// TIA Portal project "VISU_Registerlager_Template" (V14)

(* hardware
DEVICE "S7300/ET200M-Station_1"  S7-300 station
   slot 0: "Profilschiene_0"  Rail  6ES7 390-1***0-0AA0
   slot 2: "PLC_1"  CPU 315-2 PN/DP  6ES7 315-2EH13-0AB0  V2.6
      slot 1: "MPI/DP-Schnittstelle_1"  X1
      slot 2: "PROFINET-Schnittstelle_1"  PN-IO
         slot 1: "Port_1"  Port
*)

// ===== PLC "PLC_1"  CPU 315-2 PN/DP =====

VAR_GLOBAL   // PLC tag table "Standard-Variablentabelle"
   "CHAIN_REGISTER" AT %I10.0 : Bool;   // Förderkette Registerlager
   "REGISTER_ENGAGED" AT %I10.1 : Bool;   // Registerlager belegt
   "BELT_ENGAGED" AT %I10.2 : Bool;   // Förderband belegt
   "READ_SENSOR1" AT %I10.3 : Bool;   // Lesestation Sensor 1
   "READ_SENSOR2" AT %I10.4 : Bool;   // Lesestation Sensor 2
   "CONTROL_KEY" AT %I10.5 : Bool;   // Bedientaster
   "CHAIN_ON" AT %Q4.0 : Bool;   // Förderkette Regtisterlager an
   "LED_ON" AT %Q4.2 : Bool;   // LED an
   "BOX_NO" AT %MD1000 : DInt;   // Box-Nummer
   "BELT_ON" AT %Q4.1 : Bool;   // Förderband an
   "CON_KEY_TRIG" AT %M0.0 : Bool;   // 1 wenn Bedientaster gedrückt ist
   "CHAIN_REG_TRIG" AT %M0.1 : Bool;   // 1 wenn Sensor 3S1 aktiv wird
   "Counter_1" AT %MW1 : Int;   // Zähler für S1
   "Counter_2" AT %MW2 : Int;   // Zähler für S2
   "BELT_ENGAGED_TRIG" AT %M0.2 : Bool;   // 1 wenn der Nährungssensor aktiv ist
   "TIMER_FIN" AT %M0.3 : Bool;   // 1 wenn 15s Timer auslöst
END_VAR

ORGANIZATION_BLOCK "Main"   // OB1, FBD
TITLE = "Main Program Sweep (Cycle)"
{ S7_Optimized_Access := 'FALSE' }
VERSION : 0.1
   VAR_TEMP
      OB1_EV_CLASS : Byte;   // Bits 0-3 = 1 (Coming event), Bits 4-7 = 1 (Event class 1)
      OB1_SCAN_1 : Byte;   // 1 (Cold restart scan 1 of OB 1), 3 (Scan 2-n of OB 1)
      OB1_PRIORITY : Byte;   // Priority of OB Execution
      OB1_OB_NUMBR : Byte;   // 1 (Organization block 1, OB1)
      OB1_RESERVED_1 : Byte;   // Reserved for system
      OB1_RESERVED_2 : Byte;   // Reserved for system
      OB1_PREV_CYCLE : Int;   // Cycle time of previous OB1 scan (milliseconds)
      OB1_MIN_CYCLE : Int;   // Minimum cycle time of OB1 (milliseconds)
      OB1_MAX_CYCLE : Int;   // Maximum cycle time of OB1 (milliseconds)
      OB1_DATE_TIME : Date_And_Time;   // Date and time OB1 started
   END_VAR
   VAR_TEMP   // added for the SCL form of the ladder/FBD networks
      _w1 : Bool;
      _w2 : Bool;
   END_VAR
BEGIN

REGION Network 1: Förderkette und Förderband an
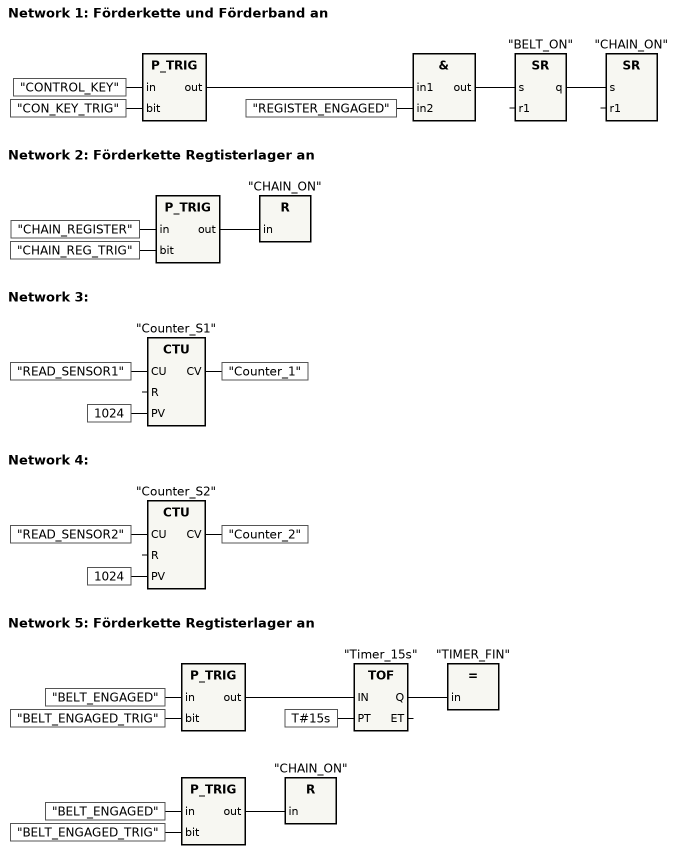
   #_w1 := "CONTROL_KEY" AND NOT "CON_KEY_TRIG";   // rising edge
   "CON_KEY_TRIG" := "CONTROL_KEY";
   IF #_w1 AND "REGISTER_ENGAGED" THEN
       "BELT_ON" := TRUE;   // SR flip-flop
   END_IF;
   IF "BELT_ON" THEN
       "CHAIN_ON" := TRUE;   // SR flip-flop
   END_IF;
END_REGION

REGION Network 2: Förderkette Regtisterlager an
   #_w1 := "CHAIN_REGISTER" AND NOT "CHAIN_REG_TRIG";   // rising edge
   "CHAIN_REG_TRIG" := "CHAIN_REGISTER";
   IF #_w1 THEN "CHAIN_ON" := FALSE; END_IF;
END_REGION

REGION Network 3
   "Counter_S1".CTU(CU := "READ_SENSOR1", PV := 1024, CV => "Counter_1");
END_REGION

REGION Network 4
   "Counter_S2".CTU(CU := "READ_SENSOR2", PV := 1024, CV => "Counter_2");
END_REGION

REGION Network 5: Förderkette Regtisterlager an
   #_w1 := "BELT_ENGAGED" AND NOT "BELT_ENGAGED_TRIG";   // rising edge
   "BELT_ENGAGED_TRIG" := "BELT_ENGAGED";
   "Timer_15s".TOF(IN := #_w1, PT := T#15s);
   "TIMER_FIN" := "Timer_15s".Q;
   #_w2 := "BELT_ENGAGED" AND NOT "BELT_ENGAGED_TRIG";   // rising edge
   "BELT_ENGAGED_TRIG" := "BELT_ENGAGED";
   IF #_w2 THEN "CHAIN_ON" := FALSE; END_IF;
END_REGION
END_ORGANIZATION_BLOCK